Universal Robots PolyScope program: cube_dev.urp

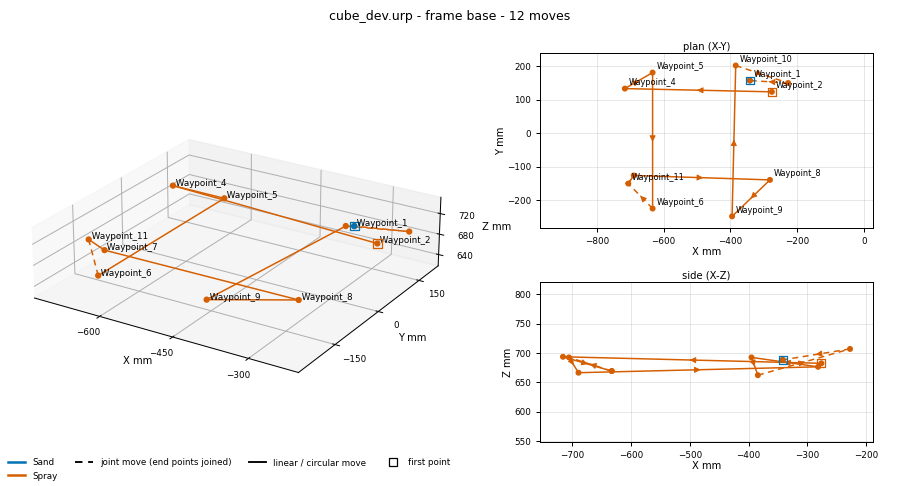
[picture p0: tool path of cube_dev.urp in frame base, 12 of 12 moves have a stored position in this frame; points joined in program order, loops and branches not executed]
Program cube_dev (installation=cube_dev directory=/programs/cube/archive createdIn=5.11.5.1010327 lastSavedIn=5.11.5.1010327 robotSerialNumber=20215500677)
Calibrated DH parameters: a=[0.000204, -0.239222, -0.391845, -0.000001, 0.000022, 0]; d=[0.162722, -355.808559, 353.37206, 2.570385, 0.099741, 0.099629]; alpha=[1.571124, 0.000988, 0.008295, 1.568963, -1.570303, 0]; deltaTheta=[0, -0.973091, 7.204745, 0.05153, 0, 0]
Robot Program (runOnlyOnce=true)
  SuppressedNode
    Wait Sleep waitTime=0.01
  Call Sand
  Call Sand
  Call Spray
  Call Spray
Event  expression=PinsBtn≟ True
  Call Spray
Event  expression=GoBtn≟ True
  Call Sand
  Call Sand
  Call Spray
  Call Spray
SubProgram -> Spray
SubProgram -> Sand
SubProgram Sand (keepSynchronizedWithDisk=false)
  Folder Sand
    MoveJ speed 60 deg/s, acceleration 80 deg/s^2 (useActiveTCP=false) tcp=SandTCP; feature=Point_1
      Waypoint Waypoint_1: TCP in base x=-341.992 y=157.901 z=688.339 mm, rx=0 ry=0 rz=-1.2285 rad; joints [-55.557, 15.2, -105.595, 194.218, -46.788, -109.717] deg; TCP offset x=3.18 y=114.64 z=98.2 mm, rx=-0.7854 ry=0 rz=0 rad; feature pose in base x=-342 y=157.897 z=730.093 mm, rx=-0.0205 ry=0.0193 rz=-1.2285 rad
    Wait Sleep waitTime=1
    MoveL speed 10 mm/s, acceleration 1200 mm/s^2 (useActiveTCP=true) feature=Base
      MoveDirectionNode (selectedDirection=ZPlus)
        Until TOOL_CONTACT_DETECTION (allowActions=false retraction=0 decelerationAcceleration=3 decelerationAngularAcceleration=34.906585)
    URCap Finishing Tool Control (Robotiq_Copilot, Robotiq Inc.) dataModel(ToolOutputNameKey=SanderOn, HackTriggeringContributionIsDefinedMethodKey=true)
    Force Simple feature=Base; selection=[0, 0, 1, 0, 0, 0]; wrench=[0, 0, 10, 0, 0, 0]; limitsForce=[0.15, 0.15, 0.15, 1.047198, 1.047198, 1.047198]; limitsMotion=[0.1, 0.1, 0.1, 0.349066, 0.349066, 0.349066]
      URCap Path Generator (Robotiq_Copilot, Robotiq Inc.) dataModel(pathOptionsTypeKey=TOOL_ON_ROBOT, PathTypeKey=FOUR_POINTS_HORIZONTAL, coverageModeKey=PERIMETER_ONLY, DimensionWidthTypeKey=FIXED, relativePathKey=true, selectedFeatureNameKey=Point_1, OriginalFeatureAsArrayKey=[-0.3029570133244077, 0.1493967343976849, 0.7821098019170267, 6.631708170368006E-5, 8.682855188236906E-5, -1.2191890682989344], offsetTypeKey=Relative to feature, PerimeterSpeedKey=100, WaypointPoseKey1=[-0.302948, 0.149426, 0.782139, 0.0206273, -0.0191894, -1.21907], WaypointJointPositionsKey1=[-0.9696818083978345, 0.1643318235311506, -1.7653774636450477, 3.4131319086056275, -0.8163088811636747, -1.9149801840548157], WaypointPoseKey3=[-0.644922, 0.149365, 0.782046, 0.0206481, -0.019077, -1.21892], WaypointJointPositionsKey3=[-0.49095242095851876, -0.11964454499745258, -0.571901094324855, 2.8481010787858114, -1.022083314926732, -2.467483944559792], WaypointPoseKey4=[-0.63206, -0.201042, 0.782555, 0.0206969, -0.0191869, -1.21902], WaypointJointPositionsKey4=[0.051157235662034665, -0.019880992789182983, -0.7779939813134202, 3.1307370565473853, -1.3661157184512103, -2.9213350582874886], WaypointPoseKey2=[-0.264867, -0.201127, 0.782458, -0.0171866, -0.0243281, 1.64706], WaypointJointPositionsKey2=[0.17181031442909458, -0.06573297505594056, -1.402976410563606, 2.256973662305123, -1.504166608950353, -0.06693468453722673], urcapVersion=1.22.1); state(isChildrenLocked=true)
        URCap Point (Robotiq_Copilot, Robotiq Inc.) dataModel(pose=[-0.302948, 0.149426, 0.782139, 0.0206273, -0.0191894, -1.21907], joint_positions=[-0.9696818083978345, 0.1643318235311506, -1.7653774636450477, 3.4131319086056275, -0.8163088811636747, -1.9149801840548157])
        URCap Point (Robotiq_Copilot, Robotiq Inc.) dataModel(pose=[-0.264867, -0.201127, 0.782458, -0.0171866, -0.0243281, 1.64706], joint_positions=[0.17181031442909458, -0.06573297505594056, -1.402976410563606, 2.256973662305123, -1.504166608950353, -0.06693468453722673])
        URCap Point (Robotiq_Copilot, Robotiq Inc.) dataModel(pose=[-0.644922, 0.149365, 0.782046, 0.0206481, -0.019077, -1.21892], joint_positions=[-0.49095242095851876, -0.11964454499745258, -0.571901094324855, 2.8481010787858114, -1.022083314926732, -2.467483944559792])
        URCap Point (Robotiq_Copilot, Robotiq Inc.) dataModel(pose=[-0.63206, -0.201042, 0.782555, 0.0206969, -0.0191869, -1.21902], joint_positions=[0.051157235662034665, -0.019880992789182983, -0.7779939813134202, 3.1307370565473853, -1.3661157184512103, -2.9213350582874886])
    URCap Finishing Tool Control (Robotiq_Copilot, Robotiq Inc.) dataModel(ToolOutputNameKey=SanderOn, HackTriggeringContributionIsDefinedMethodKey=true, FinishingToolStateKey=false)
    MoveL speed 250 mm/s, acceleration 1200 mm/s^2 (useActiveTCP=true) feature=Base
      MoveDirectionNode (selectedDirection=ZMinus) feature=Base
        Until DISTANCE (allowActions=false deceleration=3 distanceNodeType=STOP) Distance=0.075; motionParameters(blendRadius=0)
SubProgram Spray (keepSynchronizedWithDisk=false)
  Folder Spray
    Set NoAction tcp=SprayTCP
    MoveL speed 180 mm/s, acceleration 1200 mm/s^2 (useActiveTCP=false) tcp=SprayTCP; feature=Point_1
      Waypoint Waypoint_2: TCP in base x=-276.067 y=123.988 z=682.5 mm, rx=0.7212 ry=-1.4137 rz=-0.8052 rad; joints [-50.988, 17.163, -129.623, 250.086, -72.685, -298.468] deg; TCP offset x=-60.833 y=-97.548 z=92.018 mm, rx=0.1226 ry=1.1769 rz=2.8697 rad
      Set DigitalOutput pin=SprayerOn; digitalValue=1
      Waypoint Waypoint_4: TCP in base x=-716.081 y=133.693 z=693.624 mm, rx=0.7115 ry=-1.4483 rz=-0.7634 rad; joints [-17.427, 3.081, -46.874, 185.758, -99.18, -318.767] deg
      Set DigitalOutput pin=SprayerOn; digitalValue=0
      Waypoint Waypoint_5: TCP in base x=-633.048 y=181.69 z=669.306 mm, rx=1.5402 ry=-0.2522 rz=0.3695 rad; joints [-32.88, -17.39, -13.132, 100.686, -47.249, -210.075] deg
      Set DigitalOutput pin=SprayerOn; digitalValue=1
      Waypoint Waypoint_6: motionParameters(blendRadius=0.05); TCP in base x=-632.991 y=-225.358 z=669.353 mm, rx=1.5402 ry=-0.2521 rz=0.3694 rad; joints [2.928, -1.13, -39.728, 146.782, -45.925, -260.027] deg
      Set DigitalOutput pin=SprayerOn; digitalValue=0
    MoveJ speed 60 deg/s, acceleration 80 deg/s^2 (useActiveTCP=true positionType=JointAngles) feature=Base
      Waypoint Waypoint_11: TCP in base x=-705.785 y=-150.622 z=692.546 mm, rx=1.6603 ry=0.7065 rz=1.6076 rad; joints [-4.649, 6.051, -55.354, 271.275, 66.825, -330.102] deg; TCP offset x=-60.833 y=-97.548 z=92.018 mm, rx=0.1226 ry=1.1769 rz=2.8697 rad
    MoveL speed 180 mm/s, acceleration 1200 mm/s^2 (useActiveTCP=false) tcp=SprayTCP; feature=Point_1
      Waypoint Waypoint_7: TCP in base x=-689.635 y=-126.349 z=666.53 mm, rx=1.6158 ry=0.8636 rz=1.6117 rad; joints [-4.944, 10.155, -59.222, 269.746, 74.231, -329.413] deg; TCP offset x=-60.833 y=-97.548 z=92.018 mm, rx=0.1226 ry=1.1769 rz=2.8697 rad; feature pose in base x=-342 y=157.897 z=730.093 mm, rx=-0.0205 ry=0.0193 rz=-1.2285 rad
      Set DigitalOutput pin=SprayerOn; digitalValue=1
      Waypoint Waypoint_8: TCP in base x=-281.693 y=-139.617 z=676.533 mm, rx=1.6184 ry=0.8385 rz=1.6155 rad; joints [-9.325, 18.38, -130.3, 332.113, 76.22, -326.026] deg
      Set DigitalOutput pin=SprayerOn; digitalValue=0
      Waypoint Waypoint_9: TCP in base x=-395.086 y=-248.751 z=692.565 mm, rx=-0.7915 ry=-1.8187 rz=-1.9759 rad; joints [17.805, 18.205, -98.032, 302.859, 116.569, -287.675] deg; TCP offset x=-60.833 y=-97.548 z=92.018 mm, rx=0.1226 ry=1.1769 rz=2.8697 rad
      Set DigitalOutput pin=SprayerOn; digitalValue=1
      Waypoint Waypoint_10: TCP in base x=-384.214 y=202.738 z=662.283 mm, rx=-0.8556 ry=-1.8323 rz=-1.9199 rad; joints [-33.288, 14.252, -108.85, 355.917, 145.162, -229.694] deg; TCP offset x=-60.833 y=-97.548 z=92.018 mm, rx=0.1226 ry=1.1769 rz=2.8697 rad
      Set DigitalOutput pin=SprayerOn; digitalValue=0
      SuppressedNode
        MoveDirectionNode (selectedDirection=ZMinus) feature=Base
          Until DISTANCE (allowActions=false deceleration=3 distanceNodeType=STOP) Distance=0.025; motionParameters(blendRadius=0)
    MoveJ speed 60 deg/s, acceleration 80 deg/s^2 (useActiveTCP=false) tcp=SandTCP; feature=Point_1
      Waypoint Waypoint_3: TCP in base x=-227.296 y=150.39 z=706.971 mm, rx=0.0042 ry=-0.0226 rz=0.5559 rad; joints [-62.251, 12.398, -131.266, 343.992, 92.157, -175.837] deg; TCP offset x=3.18 y=114.64 z=98.2 mm, rx=-0.7854 ry=0 rz=0 rad
      Waypoint Waypoint_1: TCP in base x=-341.992 y=157.901 z=688.339 mm, rx=0 ry=0 rz=-1.2285 rad; joints [-55.557, 15.2, -105.595, 194.218, -46.788, -109.717] deg
